(* Logix 5000 project; controller PRG_SPECK Emulate 5570 rev 30.12; software revision 30.00 *)

TASK MainTask (continuous, watchdog 5000 ms) : MainProgram

MODULES
   Local : Emulate 5570 (ICP 3, rev 30.12)
       : vendor 1 type 0 code 15 (ICP 0, rev 1.1, Output RPI 50 ms)
END_MODULES

TYPE UDT_BA :
STRUCT
   AL : BOOL;
END_STRUCT
END_TYPE

PROGRAM MainProgram   (* main routine MainRoutine *)
VAR
   PRG_Counter : DINT[2];
   PRG_i : DINT;
   PRG_j : DINT;
   PRG_Res_Len : DINT;
   PRG_Result : DINT[256];
   SCAN_CYCLE_TIME : DINT;
   Speck_AS_res : DINT[2];
   Speck_AS_tmp : DINT;
   Speck_AS_X : DINT[2] := ([0] := -536870912);
   Speck_AS_Y : DINT[2] := ([0] := 1610612736);
   Speck_Block_size : DINT;
   Speck_Carry_Bit : DINT;
   Speck_Ciphertext : DINT[2,2];
   Speck_dec_i : DINT;
   Speck_dec_j : DINT;
   Speck_enc_i : DINT;
   Speck_enc_j : DINT;
   Speck_i : DINT;
   Speck_j : DINT;
   Speck_key_size : DINT;
   Speck_Plaintext : DINT[2,2];
   Speck_Rd_Max : DINT;
   Speck_Rotate_Result : DINT[2];
   Speck_Round_Keys : DINT[34,2];
   Speck_Sign_Bits : DINT[2];
   Speck_tmp : DINT;
   Speck_tmp1 : DINT;
   Speck_tmp2 : DINT[2];
   Speck_Ver : DINT;
   Speck_x : DINT[2];
   Speck_y : DINT[2];
END_VAR

ROUTINE MainRoutine   (* ladder *)
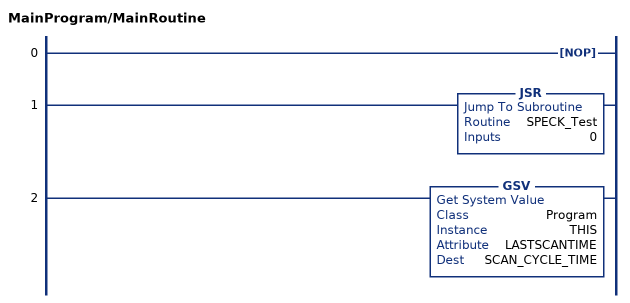
   0: NOP();
   1: JSR(SPECK_Test,0);
   2: GSV(Program,THIS,LASTSCANTIME,SCAN_CYCLE_TIME);
END_ROUTINE

ROUTINE PRG_PRF_Init   (* structured text *)
   //initialize version
   
   Speck_Ver:=2;     // 0: 32/64, 1: 64: 96, 2: 64:128, 3:128/128, 4:128/192, 5: 128/256
   
   PRG_j:=0;
   PRG_Res_Len :=  (PRG_Counter[0] AND 16#0000ffff)-1;
   
   JSR(SPECK_Init);
END_ROUTINE

ROUTINE PRG_PRF_SPECK   (* structured text *)
   // init PRG_Count[0] and PRG_Count[1] during application.. for PRF.. they could be any values
   //For PRG application, PRG_Count[0] defines the output length (i.e., the number of 64-bit, e.g., 128-bit output, PRG_Count[0]:=2)
   
   
   JSR(PRG_PRF_Init);
   
   PRG_j:=0;
   For PRG_i:=0 to PRG_Res_Len by 1 do
   	Speck_Plaintext[0,0]:=PRG_Counter[0]; //Upper bits of current plaintext
   	Speck_Plaintext[1,0]:=PRG_Counter[1];  //Lower bits of current plaintext
   	JSR(SPECK_Enc);
   	PRG_Result[PRG_j]:=Speck_Ciphertext[0,0];
   	PRG_Result[PRG_j+1]:=Speck_Ciphertext[1,0];
   
   	PRG_j:=PRG_j+2;
   
   End_For;
   
   JSR(SPECK_ClearKey);
   
END_ROUTINE

ROUTINE PRG_PRF_SPECK_Test   (* structured text *)
   
   //initialize version
   If S:FS Then
   
   	PRG_Counter[0]:=5;
   	PRG_Counter[1]:=1;
   
   
   End_if;
   
   
   JSR(PRG_PRF_SPECK);
END_ROUTINE

ROUTINE SPECK_Add   (* structured text *)
   	//big addition low 32-bit
   Speck_AS_res[0]:=0;
   Speck_AS_res[1]:=0;
   		Speck_Sign_Bits[0].[0]:= Speck_AS_X[0].30; //keep the sign bit for big addition
   		Speck_Sign_Bits[0].[1]:= Speck_AS_X[0].31;
   		Speck_AS_X[0].31:=0;
   		Speck_AS_X[0].30:=0;
   
   
   
   		Speck_Sign_Bits[1].[0]:= Speck_AS_Y[0].30; //keep the sign bit for big addition
   		Speck_Sign_Bits[1].[1]:= Speck_AS_Y[0].31;
   		Speck_AS_Y[0].31:=0;
   		Speck_AS_Y[0].30:=0;
   
   		Speck_AS_res[0] := Speck_AS_X[0]+Speck_AS_Y[0];
   
   		Speck_Carry_Bit.[0]:= Speck_AS_res[0].30;
   
   		Speck_AS_tmp:=Speck_Sign_Bits[1]+Speck_Sign_Bits[0]+Speck_Carry_Bit;
   
   		Speck_AS_res[0].[30]:= Speck_AS_tmp.[0];
   		Speck_AS_res[0].[31]:= Speck_AS_tmp.[1];
   
   		Speck_Carry_Bit.[0]:= Speck_AS_tmp.[2];
   
   
   		Speck_AS_tmp:=0;
   		Speck_Sign_Bits[0]:=0;
   		Speck_Sign_Bits[1]:=0;
   
   //add high 32-bit
   if Speck_Ver>2 then
   		Speck_Sign_Bits[0].[0]:= Speck_AS_X[1].30; //keep the sign bit for big addition
   		Speck_Sign_Bits[0].[1]:= Speck_AS_X[1].31;
   		Speck_AS_X[1].31:=0;
   		Speck_AS_X[1].30:=0;
   
   
   
   		Speck_Sign_Bits[1].[0]:= Speck_AS_Y[1].30; //keep the sign bit for big addition
   		Speck_Sign_Bits[1].[1]:= Speck_AS_Y[1].31;
   		Speck_AS_Y[1].31:=0;
   		Speck_AS_Y[1].30:=0;
   
   
   		Speck_AS_res[1]:=Speck_AS_X[1]+Speck_AS_Y[1]+Speck_Carry_Bit;
   
   		Speck_Carry_Bit.[0]:= Speck_AS_res[1].30;
   
   		Speck_AS_tmp:=Speck_Sign_Bits[1]+Speck_Sign_Bits[0]+Speck_Carry_Bit;
   
   		Speck_AS_res[1].[30]:= Speck_AS_tmp.[0];
   		Speck_AS_res[1].[31]:= Speck_AS_tmp.[1];
   
   end_if;
   
   
   		//clear
   		Speck_Carry_Bit:=0;
   		Speck_AS_tmp:=0;
   		Speck_Sign_Bits[0]:=0;
   		Speck_Sign_Bits[1]:=0;
   		Speck_AS_X[0]:=0;
   		Speck_AS_X[1]:=0;
   		Speck_AS_Y[0]:=0;
   		Speck_AS_Y[1]:=0;
   
   
END_ROUTINE

ROUTINE SPECK_ClearKey   (* structured text *)
   
   Speck_Round_Keys[0,0]:=0;
   Speck_Round_Keys[1,0]:=0;
   Speck_Round_Keys[2,0]:=0;
   Speck_Round_Keys[3,0]:=0;
   Speck_Round_Keys[4,0]:=0;
   Speck_Round_Keys[5,0]:=0;
   Speck_Round_Keys[6,0]:=0;
   Speck_Round_Keys[7,0]:=0;
   Speck_Round_Keys[8,0]:=0;
   Speck_Round_Keys[9,0]:=0;
   Speck_Round_Keys[10,0]:=0;
   Speck_Round_Keys[11,0]:=0;
   Speck_Round_Keys[12,0]:=0;
   Speck_Round_Keys[13,0]:=0;
   Speck_Round_Keys[14,0]:=0;
   Speck_Round_Keys[15,0]:=0;
   Speck_Round_Keys[16,0]:=0;
   Speck_Round_Keys[17,0]:=0;
   Speck_Round_Keys[18,0]:=0;
   Speck_Round_Keys[19,0]:=0;
   Speck_Round_Keys[20,0]:=0;
   Speck_Round_Keys[21,0]:=0;
   Speck_Round_Keys[22,0]:=0;
   Speck_Round_Keys[23,0]:=0;
   Speck_Round_Keys[24,0]:=0;
   Speck_Round_Keys[25,0]:=0;
   Speck_Round_Keys[26,0]:=0;
END_ROUTINE

ROUTINE SPECK_Dec   (* structured text *)
   
   JSR(SPECK_Init);
   
   
   
   
   Case Speck_Ver Of
   
   0,1,2:
   	Speck_Plaintext[0,0]:=Speck_Ciphertext[0,0];
   	Speck_Plaintext[1,0]:=Speck_Ciphertext[1,0];
   
   	For Speck_i:=Speck_Rd_Max to 0 by -1 do
   
   		Speck_AS_res[0]:= Speck_Plaintext[1,0] XOR Speck_Plaintext[0,0];
   
   		Speck_tmp2[0]:=Speck_AS_res[0];
   		JSR(SPECK_Rotate_Right_Dec);      //rotate based on Speck_AS_res[0]
   
   		Speck_Plaintext[0,0]:= Speck_Rotate_Result[0];
   
   		Speck_AS_X[0]:= Speck_Plaintext[1,0] XOR Speck_Round_Keys[Speck_i,0];
   
   
   
   		if Speck_Ver=0 Then
   			Speck_AS_X[0].16:=1;
   			Speck_AS_res[0]:= (Speck_AS_X[0]- Speck_Plaintext[0,0]) AND 16#0000ffff; //??AND 16#ffff;
   		Else
   			Speck_AS_Y[0]:=Speck_Plaintext[0,0];
   			JSR(SPECK_Sub);
   		End_if;
   		Speck_tmp2[0]:=Speck_AS_res[0];
   		JSR(SPECK_Rotate_Left_Dec);      //rotate based on Speck_AS_res[0]
   		Speck_Plaintext[1,0]:=Speck_Rotate_Result[0];
   
   	End_for;
   
   3,4,5:
   	Speck_Plaintext[0,0]:=Speck_Ciphertext[0,0];
   	Speck_Plaintext[0,1]:=Speck_Ciphertext[0,1];
   	Speck_Plaintext[1,0]:=Speck_Ciphertext[1,0];
   	Speck_Plaintext[1,1]:=Speck_Ciphertext[1,1];
   
   	For Speck_i:=Speck_Rd_Max to 0 by -1 do
   
   		Speck_AS_res[0]:= Speck_Plaintext[0,0] XOR Speck_Plaintext[1,0];
   		Speck_AS_res[1]:= Speck_Plaintext[0,1] XOR Speck_Plaintext[1,1];
   
   
   		Speck_tmp2[0]:=Speck_AS_res[0];
   		Speck_tmp2[1]:=Speck_AS_res[1];
   		JSR(SPECK_Rotate_Right_Dec);      //rotate based on Speck_AS_res[0] and Speck_AS_res[1]
   
   		Speck_Plaintext[0,0]:= Speck_Rotate_Result[0];
   		Speck_Plaintext[0,1]:= Speck_Rotate_Result[1];
   
   		Speck_AS_X[0]:= Speck_Plaintext[1,0] XOR Speck_Round_Keys[Speck_i,0];
   		Speck_AS_X[1]:= Speck_Plaintext[1,1] XOR Speck_Round_Keys[Speck_i,1];
   
   
   		Speck_AS_Y[0]:=Speck_Plaintext[0,0];
   		Speck_AS_Y[1]:=Speck_Plaintext[0,1];
   		JSR(SPECK_Sub);
   
   		Speck_tmp2[0]:=Speck_AS_res[0];
   		Speck_tmp2[1]:=Speck_AS_res[1];
   		JSR(SPECK_Rotate_Left_Dec);      //rotate based on Speck_AS_res[0] and Speck_AS_res[1]
   		Speck_Plaintext[1,0]:=Speck_Rotate_Result[0];
   		Speck_Plaintext[1,1]:=Speck_Rotate_Result[1];
   	End_for;
   
   End_Case;
   
   
   
   
   
   
   JSR(SPECK_ClearKey);
   
   
   
   
   
   
   
   
END_ROUTINE

ROUTINE SPECK_Enc   (* structured text *)
   
   Case Speck_Ver Of
   
   0,1,2:
   	Speck_Ciphertext[0,0]:=Speck_Plaintext[0,0];
   	Speck_Ciphertext[1,0]:=Speck_Plaintext[1,0];
   
   	For Speck_i:=0 to Speck_Rd_Max by 1 do
   		Speck_tmp2[0]:=Speck_Ciphertext[1,0];
   		JSR(SPECK_Rotate_Right_Enc);       //c1>>>>
   
   
   
   
   		if Speck_Ver=0 Then
   			Speck_Ciphertext[1,0]:= (Speck_Rotate_Result[0] + Speck_Ciphertext[0,0]) XOR Speck_Round_Keys[Speck_i,0];
   			Speck_Ciphertext[1,0]:= Speck_Ciphertext[1,0] AND 16#0000ffff;
   		Else
   			Speck_AS_X[0]:=Speck_Rotate_Result[0];
   			Speck_AS_Y[0]:=Speck_Ciphertext[0,0];
   			JSR(SPECK_Add);
   			Speck_Ciphertext[1,0]:= Speck_AS_res[0] XOR Speck_Round_Keys[Speck_i,0];
   		End_if;
   
   
   		Speck_tmp2[0]:=Speck_Ciphertext[0,0];
   		JSR(SPECK_Rotate_Left_Enc);   //p0<<<
   		Speck_Ciphertext[0,0]:=Speck_Rotate_Result[0] XOR Speck_Ciphertext[1,0];
   	End_for;
   
   3,4,5:
   	Speck_Ciphertext[0,0]:=Speck_Plaintext[0,0];
   	Speck_Ciphertext[0,1]:=Speck_Plaintext[0,1];
   	Speck_Ciphertext[1,0]:=Speck_Plaintext[1,0];
   	Speck_Ciphertext[1,1]:=Speck_Plaintext[1,1];
   
   	For Speck_i:=0 to Speck_Rd_Max by 1 do
   		Speck_tmp2[0]:=Speck_Ciphertext[1,0];
   		Speck_tmp2[1]:=Speck_Ciphertext[1,1];
   		JSR(SPECK_Rotate_Right_Enc);       //c1>>>>
   
   
   
   
   		Speck_AS_X[0]:=Speck_Rotate_Result[0];
   		Speck_AS_X[1]:=Speck_Rotate_Result[1];
   		Speck_AS_Y[0]:=Speck_Ciphertext[0,0];
   		Speck_AS_Y[1]:=Speck_Ciphertext[0,1];
   		JSR(SPECK_Add);
   		Speck_Ciphertext[1,0]:= Speck_AS_res[0] XOR Speck_Round_Keys[Speck_i,0];
   	 	Speck_Ciphertext[1,1]:= Speck_AS_res[1] XOR Speck_Round_Keys[Speck_i,1];
   
   
   		Speck_tmp2[0]:=Speck_Ciphertext[0,0];
   		Speck_tmp2[1]:=Speck_Ciphertext[0,1];
   		JSR(SPECK_Rotate_Left_Enc);   //c0<<<
   		Speck_Ciphertext[0,0]:=Speck_Rotate_Result[0] XOR Speck_Ciphertext[1,0];
   		Speck_Ciphertext[0,1]:=Speck_Rotate_Result[1] XOR Speck_Ciphertext[1,1];
   	End_for;
   
   End_Case;
   
   
   
   
   
   JSR(SPECK_ClearKey);
   
   
   
   
   
   
END_ROUTINE

ROUTINE SPECK_Init   (* structured text *)
   CASE Speck_Ver Of
   	0:
   		//Speck_Rd_Max:=21;
   		Speck_Rd_Max:=21;
   		Speck_Round_Keys[0,0]:=15631;
   		//Speck_Round_Keys[0,0]:=0;
   		Speck_Round_Keys[1,0]:=9700;
   		Speck_Round_Keys[2,0]:=61996;
   		Speck_Round_Keys[3,0]:=19213;
   		Speck_Round_Keys[4,0]:=12568;
   		Speck_Round_Keys[5,0]:=53935;
   		Speck_Round_Keys[6,0]:=268;
   		Speck_Round_Keys[7,0]:=50664;
   		Speck_Round_Keys[8,0]:=60120;
   		Speck_Round_Keys[9,0]:=40333;
   		Speck_Round_Keys[10,0]:=24732;
   		Speck_Round_Keys[11,0]:=23055;
   		Speck_Round_Keys[12,0]:=43006;
   		Speck_Round_Keys[13,0]:=3801;
   		Speck_Round_Keys[14,0]:=54139;
   		Speck_Round_Keys[15,0]:=30112;
   		Speck_Round_Keys[16,0]:=55913;
   		Speck_Round_Keys[17,0]:=28143;
   		Speck_Round_Keys[18,0]:=63915;
   		Speck_Round_Keys[19,0]:=1151;
   		Speck_Round_Keys[20,0]:=48927;
   		Speck_Round_Keys[21,0]:=23424;
   	1:
   		Speck_Rd_Max:=25;
   		Speck_Round_Keys[0,0]:=1010479052;
   		Speck_Round_Keys[1,0]:=1960303416;
   		Speck_Round_Keys[2,0]:=1299975900;
   		Speck_Round_Keys[3,0]:=-1898951853;
   		Speck_Round_Keys[4,0]:=-1343771839;
   		Speck_Round_Keys[5,0]:=1072967228;
   		Speck_Round_Keys[6,0]:=1891935448;
   		Speck_Round_Keys[7,0]:=-862191615;
   		Speck_Round_Keys[8,0]:=-24294679;
   		Speck_Round_Keys[9,0]:=1209777;
   		Speck_Round_Keys[10,0]:=-379647130;
   		Speck_Round_Keys[11,0]:=-429531458;
   		Speck_Round_Keys[12,0]:=1219013850;
   		Speck_Round_Keys[13,0]:=1258773305;
   		Speck_Round_Keys[14,0]:=1958978832;
   		Speck_Round_Keys[15,0]:=-1299080388;
   		Speck_Round_Keys[16,0]:=1521232504;
   		Speck_Round_Keys[17,0]:=-1755465132;
   		Speck_Round_Keys[18,0]:=-1183209214;
   		Speck_Round_Keys[19,0]:=-497510761;
   		Speck_Round_Keys[20,0]:=-65018188;
   		Speck_Round_Keys[21,0]:=627271131;
   		Speck_Round_Keys[22,0]:=289351083;
   		Speck_Round_Keys[23,0]:=163990315;
   		Speck_Round_Keys[24,0]:=-1174022665;
   		Speck_Round_Keys[25,0]:=-1342639090;
   	2:
   		Speck_Rd_Max:=26;
   		Speck_Round_Keys[0,0]:=-1148848103;
   		Speck_Round_Keys[1,0]:=1208089977;
   		Speck_Round_Keys[2,0]:=-1783362989;
   		Speck_Round_Keys[3,0]:=-914269261;
   		Speck_Round_Keys[4,0]:=-1304315992;
   		Speck_Round_Keys[5,0]:=-2127551690;
   		Speck_Round_Keys[6,0]:=-823047894;
   		Speck_Round_Keys[7,0]:=-1124290961;
   		Speck_Round_Keys[8,0]:=-2081609188;
   		Speck_Round_Keys[9,0]:=-1368174669;
   		Speck_Round_Keys[10,0]:=1254090106;
   		Speck_Round_Keys[11,0]:=-1215402569;
   		Speck_Round_Keys[12,0]:=-1522370332;
   		Speck_Round_Keys[13,0]:=-9254945;
   		Speck_Round_Keys[14,0]:=-770318043;
   		Speck_Round_Keys[15,0]:=-1248627894;
   		Speck_Round_Keys[16,0]:=1667665164;
   		Speck_Round_Keys[17,0]:=1127551330;
   		Speck_Round_Keys[18,0]:=1631463370;
   		Speck_Round_Keys[19,0]:=339858424;
   		Speck_Round_Keys[20,0]:=1104564693;
   		Speck_Round_Keys[21,0]:=-1092140090;
   		Speck_Round_Keys[22,0]:=-34819784;
   		Speck_Round_Keys[23,0]:=-1239678853;
   		Speck_Round_Keys[24,0]:=1539057967;
   		Speck_Round_Keys[25,0]:=1646443297;
   		Speck_Round_Keys[26,0]:=99633891;
   	3:
   		Speck_Rd_Max:=31;
   		Speck_Round_Keys[0,0]:=-2080825868;
   		Speck_Round_Keys[0,1]:=-649265456;
   		Speck_Round_Keys[1,0]:=2050826354;
   		Speck_Round_Keys[1,1]:=789043958;
   		Speck_Round_Keys[2,0]:=1076159464;
   		Speck_Round_Keys[2,1]:=1207346796;
   		Speck_Round_Keys[3,0]:=-1868617995;
   		Speck_Round_Keys[3,1]:=27785654;
   		Speck_Round_Keys[4,0]:=653389667;
   		Speck_Round_Keys[4,1]:=857678648;
   		Speck_Round_Keys[5,0]:=1480341691;
   		Speck_Round_Keys[5,1]:=-1263296287;
   		Speck_Round_Keys[6,0]:=-1964153065;
   		Speck_Round_Keys[6,1]:=-1671577777;
   		Speck_Round_Keys[7,0]:=862328600;
   		Speck_Round_Keys[7,1]:=2036511554;
   		Speck_Round_Keys[8,0]:=81192154;
   		Speck_Round_Keys[8,1]:=-687588873;
   		Speck_Round_Keys[9,0]:=-1917483227;
   		Speck_Round_Keys[9,1]:=63249243;
   		Speck_Round_Keys[10,0]:=-1952596082;
   		Speck_Round_Keys[10,1]:=2143544786;
   		Speck_Round_Keys[11,0]:=-1544920938;
   		Speck_Round_Keys[11,1]:=1465879784;
   		Speck_Round_Keys[12,0]:=2139891583;
   		Speck_Round_Keys[12,1]:=1710163122;
   		Speck_Round_Keys[13,0]:=-1608051307;
   		Speck_Round_Keys[13,1]:=-1374801591;
   		Speck_Round_Keys[14,0]:=943121719;
   		Speck_Round_Keys[14,1]:=354429694;
   		Speck_Round_Keys[15,0]:=582741445;
   		Speck_Round_Keys[15,1]:=-2054972675;
   		Speck_Round_Keys[16,0]:=1721968636;
   		Speck_Round_Keys[16,1]:=-1512022332;
   		Speck_Round_Keys[17,0]:=-1725680323;
   		Speck_Round_Keys[17,1]:=1657126074;
   		Speck_Round_Keys[18,0]:=247339174;
   		Speck_Round_Keys[18,1]:=1221108278;
   		Speck_Round_Keys[19,0]:=-807872440;
   		Speck_Round_Keys[19,1]:=-1429436100;
   		Speck_Round_Keys[20,0]:=1418166873;
   		Speck_Round_Keys[20,1]:=-215130835;
   		Speck_Round_Keys[21,0]:=-621280229;
   		Speck_Round_Keys[21,1]:=412315805;
   		Speck_Round_Keys[22,0]:=1459956154;
   		Speck_Round_Keys[22,1]:=-1758754260;
   		Speck_Round_Keys[23,0]:=435300123;
   		Speck_Round_Keys[23,1]:=-1545364290;
   		Speck_Round_Keys[24,0]:=1027574508;
   		Speck_Round_Keys[24,1]:=-481319156;
   		Speck_Round_Keys[25,0]:=1691703329;
   		Speck_Round_Keys[25,1]:=651500257;
   		Speck_Round_Keys[26,0]:=1740505566;
   		Speck_Round_Keys[26,1]:=1823342560;
   		Speck_Round_Keys[27,0]:=1022031660;
   		Speck_Round_Keys[27,1]:=749650446;
   		Speck_Round_Keys[28,0]:=-397311955;
   		Speck_Round_Keys[28,1]:=83994786;
   		Speck_Round_Keys[29,0]:=800982389;
   		Speck_Round_Keys[29,1]:=-646252930;
   		Speck_Round_Keys[30,0]:=1439684980;
   		Speck_Round_Keys[30,1]:=386814096;
   		Speck_Round_Keys[31,0]:=-873348581;
   		Speck_Round_Keys[31,1]:=-1190976360;
   	4:
   		Speck_Rd_Max:=32;
   		Speck_Round_Keys[0,0]:=-2109044216;
   		Speck_Round_Keys[0,1]:=-434844049;
   		Speck_Round_Keys[1,0]:=-1420570460;
   		Speck_Round_Keys[1,1]:=2000435062;
   		Speck_Round_Keys[2,0]:=663289456;
   		Speck_Round_Keys[2,1]:=-1180846514;
   		Speck_Round_Keys[3,0]:=1579651993;
   		Speck_Round_Keys[3,1]:=66732943;
   		Speck_Round_Keys[4,0]:=-949825977;
   		Speck_Round_Keys[4,1]:=-1943390162;
   		Speck_Round_Keys[5,0]:=586375629;
   		Speck_Round_Keys[5,1]:=992192424;
   		Speck_Round_Keys[6,0]:=805843267;
   		Speck_Round_Keys[6,1]:=1590578209;
   		Speck_Round_Keys[7,0]:=-1864178662;
   		Speck_Round_Keys[7,1]:=-488374217;
   		Speck_Round_Keys[8,0]:=1152511586;
   		Speck_Round_Keys[8,1]:=-194034418;
   		Speck_Round_Keys[9,0]:=-916674430;
   		Speck_Round_Keys[9,1]:=510305946;
   		Speck_Round_Keys[10,0]:=61438023;
   		Speck_Round_Keys[10,1]:=-443574147;
   		Speck_Round_Keys[11,0]:=1283870034;
   		Speck_Round_Keys[11,1]:=1171556711;
   		Speck_Round_Keys[12,0]:=-1044183024;
   		Speck_Round_Keys[12,1]:=1485368022;
   		Speck_Round_Keys[13,0]:=60705369;
   		Speck_Round_Keys[13,1]:=1673274192;
   		Speck_Round_Keys[14,0]:=181714170;
   		Speck_Round_Keys[14,1]:=-810971494;
   		Speck_Round_Keys[15,0]:=-1452546250;
   		Speck_Round_Keys[15,1]:=-2049570575;
   		Speck_Round_Keys[16,0]:=563980564;
   		Speck_Round_Keys[16,1]:=1508672253;
   		Speck_Round_Keys[17,0]:=-1726885166;
   		Speck_Round_Keys[17,1]:=1988838192;
   		Speck_Round_Keys[18,0]:=-11526877;
   		Speck_Round_Keys[18,1]:=-1858736650;
   		Speck_Round_Keys[19,0]:=-963990845;
   		Speck_Round_Keys[19,1]:=-817492171;
   		Speck_Round_Keys[20,0]:=1478577398;
   		Speck_Round_Keys[20,1]:=-1380080500;
   		Speck_Round_Keys[21,0]:=-1676330340;
   		Speck_Round_Keys[21,1]:=1534823287;
   		Speck_Round_Keys[22,0]:=-2026497924;
   		Speck_Round_Keys[22,1]:=-1854221332;
   		Speck_Round_Keys[23,0]:=1666823377;
   		Speck_Round_Keys[23,1]:=1853488750;
   		Speck_Round_Keys[24,0]:=-158124369;
   		Speck_Round_Keys[24,1]:=-1736367530;
   		Speck_Round_Keys[25,0]:=1832056096;
   		Speck_Round_Keys[25,1]:=-709491608;
   		Speck_Round_Keys[26,0]:=-1320038234;
   		Speck_Round_Keys[26,1]:=-946880541;
   		Speck_Round_Keys[27,0]:=-2048989650;
   		Speck_Round_Keys[27,1]:=1069091871;
   		Speck_Round_Keys[28,0]:=-1081468659;
   		Speck_Round_Keys[28,1]:=493915857;
   		Speck_Round_Keys[29,0]:=1244604632;
   		Speck_Round_Keys[29,1]:=209165789;
   		Speck_Round_Keys[30,0]:=-516878538;
   		Speck_Round_Keys[30,1]:=967074394;
   		Speck_Round_Keys[31,0]:=528572285;
   		Speck_Round_Keys[31,1]:=-27129480;
   		Speck_Round_Keys[32,0]:=-1066840277;
   		Speck_Round_Keys[32,1]:=-1998704319;
   	5:
   		Speck_Rd_Max:=33;
   		//Speck_Rd_Max:=0;
   		Speck_Round_Keys[0,0]:=-1203303343;
   		Speck_Round_Keys[0,1]:=1330976216;
   		Speck_Round_Keys[1,0]:=1407326483;
   		Speck_Round_Keys[1,1]:=-1724620941;
   		Speck_Round_Keys[2,0]:=-1336357073;
   		Speck_Round_Keys[2,1]:=2075201973;
   		Speck_Round_Keys[3,0]:=-1964127817;
   		Speck_Round_Keys[3,1]:=-1676860110;
   		Speck_Round_Keys[4,0]:=-2129443066;
   		Speck_Round_Keys[4,1]:=1324272631;
   		Speck_Round_Keys[5,0]:=-1616999486;
   		Speck_Round_Keys[5,1]:=1032033716;
   		Speck_Round_Keys[6,0]:=238450941;
   		Speck_Round_Keys[6,1]:=454117302;
   		Speck_Round_Keys[7,0]:=-2133053345;
   		Speck_Round_Keys[7,1]:=2016900436;
   		Speck_Round_Keys[8,0]:=1979592355;
   		Speck_Round_Keys[8,1]:=-1585551365;
   		Speck_Round_Keys[9,0]:=1247927760;
   		Speck_Round_Keys[9,1]:=559820155;
   		Speck_Round_Keys[10,0]:=2074240269;
   		Speck_Round_Keys[10,1]:=1096187537;
   		Speck_Round_Keys[11,0]:=-1544710491;
   		Speck_Round_Keys[11,1]:=-971052382;
   		Speck_Round_Keys[12,0]:=1614561484;
   		Speck_Round_Keys[12,1]:=-1118146933;
   		Speck_Round_Keys[13,0]:=625176544;
   		Speck_Round_Keys[13,1]:=-1517436671;
   		Speck_Round_Keys[14,0]:=-1440617253;
   		Speck_Round_Keys[14,1]:=-1662713437;
   		Speck_Round_Keys[15,0]:=503283530;
   		Speck_Round_Keys[15,1]:=1995145044;
   		Speck_Round_Keys[16,0]:=284729323;
   		Speck_Round_Keys[16,1]:=-825926335;
   		Speck_Round_Keys[17,0]:=1430104656;
   		Speck_Round_Keys[17,1]:=-1991245376;
   		Speck_Round_Keys[18,0]:=294868347;
   		Speck_Round_Keys[18,1]:=-458348607;
   		Speck_Round_Keys[19,0]:=1158525600;
   		Speck_Round_Keys[19,1]:=601377666;
   		Speck_Round_Keys[20,0]:=1936684124;
   		Speck_Round_Keys[20,1]:=1623592388;
   		Speck_Round_Keys[21,0]:=1182373476;
   		Speck_Round_Keys[21,1]:=795858385;
   		Speck_Round_Keys[22,0]:=-1645874420;
   		Speck_Round_Keys[22,1]:=755343120;
   		Speck_Round_Keys[23,0]:=1526816951;
   		Speck_Round_Keys[23,1]:=247936705;
   		Speck_Round_Keys[24,0]:=2013201414;
   		Speck_Round_Keys[24,1]:=-80764261;
   		Speck_Round_Keys[25,0]:=326734656;
   		Speck_Round_Keys[25,1]:=-857819692;
   		Speck_Round_Keys[26,0]:=22458222;
   		Speck_Round_Keys[26,1]:=1789592334;
   		Speck_Round_Keys[27,0]:=-53318718;
   		Speck_Round_Keys[27,1]:=2100444963;
   		Speck_Round_Keys[28,0]:=-31841512;
   		Speck_Round_Keys[28,1]:=-838605044;
   		Speck_Round_Keys[29,0]:=-1477810343;
   		Speck_Round_Keys[29,1]:=-1127145226;
   		Speck_Round_Keys[30,0]:=-1047355237;
   		Speck_Round_Keys[30,1]:=-232830838;
   		Speck_Round_Keys[31,0]:=842943118;
   		Speck_Round_Keys[31,1]:=1252680607;
   		Speck_Round_Keys[32,0]:=-1978168146;
   		Speck_Round_Keys[32,1]:=2089790505;
   		Speck_Round_Keys[33,0]:=1886440712;
   		Speck_Round_Keys[33,1]:=1660119865;
   End_CASE;
   
END_ROUTINE

ROUTINE SPECK_Rotate_Left_Dec   (* structured text *)
   Speck_Rotate_Result[0]:=0;
   Speck_Rotate_Result[1]:=0;
   
   CASE Speck_Ver Of
   	0:
   		Speck_Rotate_Result[0].[6]:=Speck_tmp2[0].[15];
   		Speck_Rotate_Result[0].[5]:=Speck_tmp2[0].[14];
   		Speck_Rotate_Result[0].[4]:=Speck_tmp2[0].[13];
   		Speck_Rotate_Result[0].[3]:=Speck_tmp2[0].[12];
   		Speck_Rotate_Result[0].[2]:=Speck_tmp2[0].[11];
   		Speck_Rotate_Result[0].[1]:=Speck_tmp2[0].[10];
   		Speck_Rotate_Result[0].[0]:=Speck_tmp2[0].[9];
   		Speck_Rotate_Result[0].[15]:=Speck_tmp2[0].[8];
   		Speck_Rotate_Result[0].[14]:=Speck_tmp2[0].[7];
   		Speck_Rotate_Result[0].[13]:=Speck_tmp2[0].[6];
   		Speck_Rotate_Result[0].[12]:=Speck_tmp2[0].[5];
   		Speck_Rotate_Result[0].[11]:=Speck_tmp2[0].[4];
   		Speck_Rotate_Result[0].[10]:=Speck_tmp2[0].[3];
   		Speck_Rotate_Result[0].[9]:=Speck_tmp2[0].[2];
   		Speck_Rotate_Result[0].[8]:=Speck_tmp2[0].[1];
   		Speck_Rotate_Result[0].[7]:=Speck_tmp2[0].[0];
   	1,2:
   		Speck_Rotate_Result[0].[7]:=Speck_tmp2[0].[31];
   		Speck_Rotate_Result[0].[6]:=Speck_tmp2[0].[30];
   		Speck_Rotate_Result[0].[5]:=Speck_tmp2[0].[29];
   		Speck_Rotate_Result[0].[4]:=Speck_tmp2[0].[28];
   		Speck_Rotate_Result[0].[3]:=Speck_tmp2[0].[27];
   		Speck_Rotate_Result[0].[2]:=Speck_tmp2[0].[26];
   		Speck_Rotate_Result[0].[1]:=Speck_tmp2[0].[25];
   		Speck_Rotate_Result[0].[0]:=Speck_tmp2[0].[24];
   		Speck_Rotate_Result[0].[31]:=Speck_tmp2[0].[23];
   		Speck_Rotate_Result[0].[30]:=Speck_tmp2[0].[22];
   		Speck_Rotate_Result[0].[29]:=Speck_tmp2[0].[21];
   		Speck_Rotate_Result[0].[28]:=Speck_tmp2[0].[20];
   		Speck_Rotate_Result[0].[27]:=Speck_tmp2[0].[19];
   		Speck_Rotate_Result[0].[26]:=Speck_tmp2[0].[18];
   		Speck_Rotate_Result[0].[25]:=Speck_tmp2[0].[17];
   		Speck_Rotate_Result[0].[24]:=Speck_tmp2[0].[16];
   		Speck_Rotate_Result[0].[23]:=Speck_tmp2[0].[15];
   		Speck_Rotate_Result[0].[22]:=Speck_tmp2[0].[14];
   		Speck_Rotate_Result[0].[21]:=Speck_tmp2[0].[13];
   		Speck_Rotate_Result[0].[20]:=Speck_tmp2[0].[12];
   		Speck_Rotate_Result[0].[19]:=Speck_tmp2[0].[11];
   		Speck_Rotate_Result[0].[18]:=Speck_tmp2[0].[10];
   		Speck_Rotate_Result[0].[17]:=Speck_tmp2[0].[9];
   		Speck_Rotate_Result[0].[16]:=Speck_tmp2[0].[8];
   		Speck_Rotate_Result[0].[15]:=Speck_tmp2[0].[7];
   		Speck_Rotate_Result[0].[14]:=Speck_tmp2[0].[6];
   		Speck_Rotate_Result[0].[13]:=Speck_tmp2[0].[5];
   		Speck_Rotate_Result[0].[12]:=Speck_tmp2[0].[4];
   		Speck_Rotate_Result[0].[11]:=Speck_tmp2[0].[3];
   		Speck_Rotate_Result[0].[10]:=Speck_tmp2[0].[2];
   		Speck_Rotate_Result[0].[9]:=Speck_tmp2[0].[1];
   		Speck_Rotate_Result[0].[8]:=Speck_tmp2[0].[0];
   	3,4,5:
   		Speck_Rotate_Result[0].[7]:=Speck_tmp2[1].[31];
   		Speck_Rotate_Result[0].[6]:=Speck_tmp2[1].[30];
   		Speck_Rotate_Result[0].[5]:=Speck_tmp2[1].[29];
   		Speck_Rotate_Result[0].[4]:=Speck_tmp2[1].[28];
   		Speck_Rotate_Result[0].[3]:=Speck_tmp2[1].[27];
   		Speck_Rotate_Result[0].[2]:=Speck_tmp2[1].[26];
   		Speck_Rotate_Result[0].[1]:=Speck_tmp2[1].[25];
   		Speck_Rotate_Result[0].[0]:=Speck_tmp2[1].[24];
   		Speck_Rotate_Result[1].[31]:=Speck_tmp2[1].[23];
   		Speck_Rotate_Result[1].[30]:=Speck_tmp2[1].[22];
   		Speck_Rotate_Result[1].[29]:=Speck_tmp2[1].[21];
   		Speck_Rotate_Result[1].[28]:=Speck_tmp2[1].[20];
   		Speck_Rotate_Result[1].[27]:=Speck_tmp2[1].[19];
   		Speck_Rotate_Result[1].[26]:=Speck_tmp2[1].[18];
   		Speck_Rotate_Result[1].[25]:=Speck_tmp2[1].[17];
   		Speck_Rotate_Result[1].[24]:=Speck_tmp2[1].[16];
   		Speck_Rotate_Result[1].[23]:=Speck_tmp2[1].[15];
   		Speck_Rotate_Result[1].[22]:=Speck_tmp2[1].[14];
   		Speck_Rotate_Result[1].[21]:=Speck_tmp2[1].[13];
   		Speck_Rotate_Result[1].[20]:=Speck_tmp2[1].[12];
   		Speck_Rotate_Result[1].[19]:=Speck_tmp2[1].[11];
   		Speck_Rotate_Result[1].[18]:=Speck_tmp2[1].[10];
   		Speck_Rotate_Result[1].[17]:=Speck_tmp2[1].[9];
   		Speck_Rotate_Result[1].[16]:=Speck_tmp2[1].[8];
   		Speck_Rotate_Result[1].[15]:=Speck_tmp2[1].[7];
   		Speck_Rotate_Result[1].[14]:=Speck_tmp2[1].[6];
   		Speck_Rotate_Result[1].[13]:=Speck_tmp2[1].[5];
   		Speck_Rotate_Result[1].[12]:=Speck_tmp2[1].[4];
   		Speck_Rotate_Result[1].[11]:=Speck_tmp2[1].[3];
   		Speck_Rotate_Result[1].[10]:=Speck_tmp2[1].[2];
   		Speck_Rotate_Result[1].[9]:=Speck_tmp2[1].[1];
   		Speck_Rotate_Result[1].[8]:=Speck_tmp2[1].[0];
   		Speck_Rotate_Result[1].[7]:=Speck_tmp2[0].[31];
   		Speck_Rotate_Result[1].[6]:=Speck_tmp2[0].[30];
   		Speck_Rotate_Result[1].[5]:=Speck_tmp2[0].[29];
   		Speck_Rotate_Result[1].[4]:=Speck_tmp2[0].[28];
   		Speck_Rotate_Result[1].[3]:=Speck_tmp2[0].[27];
   		Speck_Rotate_Result[1].[2]:=Speck_tmp2[0].[26];
   		Speck_Rotate_Result[1].[1]:=Speck_tmp2[0].[25];
   		Speck_Rotate_Result[1].[0]:=Speck_tmp2[0].[24];
   		Speck_Rotate_Result[0].[31]:=Speck_tmp2[0].[23];
   		Speck_Rotate_Result[0].[30]:=Speck_tmp2[0].[22];
   		Speck_Rotate_Result[0].[29]:=Speck_tmp2[0].[21];
   		Speck_Rotate_Result[0].[28]:=Speck_tmp2[0].[20];
   		Speck_Rotate_Result[0].[27]:=Speck_tmp2[0].[19];
   		Speck_Rotate_Result[0].[26]:=Speck_tmp2[0].[18];
   		Speck_Rotate_Result[0].[25]:=Speck_tmp2[0].[17];
   		Speck_Rotate_Result[0].[24]:=Speck_tmp2[0].[16];
   		Speck_Rotate_Result[0].[23]:=Speck_tmp2[0].[15];
   		Speck_Rotate_Result[0].[22]:=Speck_tmp2[0].[14];
   		Speck_Rotate_Result[0].[21]:=Speck_tmp2[0].[13];
   		Speck_Rotate_Result[0].[20]:=Speck_tmp2[0].[12];
   		Speck_Rotate_Result[0].[19]:=Speck_tmp2[0].[11];
   		Speck_Rotate_Result[0].[18]:=Speck_tmp2[0].[10];
   		Speck_Rotate_Result[0].[17]:=Speck_tmp2[0].[9];
   		Speck_Rotate_Result[0].[16]:=Speck_tmp2[0].[8];
   		Speck_Rotate_Result[0].[15]:=Speck_tmp2[0].[7];
   		Speck_Rotate_Result[0].[14]:=Speck_tmp2[0].[6];
   		Speck_Rotate_Result[0].[13]:=Speck_tmp2[0].[5];
   		Speck_Rotate_Result[0].[12]:=Speck_tmp2[0].[4];
   		Speck_Rotate_Result[0].[11]:=Speck_tmp2[0].[3];
   		Speck_Rotate_Result[0].[10]:=Speck_tmp2[0].[2];
   		Speck_Rotate_Result[0].[9]:=Speck_tmp2[0].[1];
   		Speck_Rotate_Result[0].[8]:=Speck_tmp2[0].[0];
   End_CASE;
   
END_ROUTINE

ROUTINE SPECK_Rotate_Left_Enc   (* structured text *)
   Speck_Rotate_Result[0]:=0;
   Speck_Rotate_Result[1]:=0;
   CASE Speck_Ver Of
   	0:
   		Speck_Rotate_Result[0].[1]:=Speck_tmp2[0].[15];
   		Speck_Rotate_Result[0].[0]:=Speck_tmp2[0].[14];
   		Speck_Rotate_Result[0].[15]:=Speck_tmp2[0].[13];
   		Speck_Rotate_Result[0].[14]:=Speck_tmp2[0].[12];
   		Speck_Rotate_Result[0].[13]:=Speck_tmp2[0].[11];
   		Speck_Rotate_Result[0].[12]:=Speck_tmp2[0].[10];
   		Speck_Rotate_Result[0].[11]:=Speck_tmp2[0].[9];
   		Speck_Rotate_Result[0].[10]:=Speck_tmp2[0].[8];
   		Speck_Rotate_Result[0].[9]:=Speck_tmp2[0].[7];
   		Speck_Rotate_Result[0].[8]:=Speck_tmp2[0].[6];
   		Speck_Rotate_Result[0].[7]:=Speck_tmp2[0].[5];
   		Speck_Rotate_Result[0].[6]:=Speck_tmp2[0].[4];
   		Speck_Rotate_Result[0].[5]:=Speck_tmp2[0].[3];
   		Speck_Rotate_Result[0].[4]:=Speck_tmp2[0].[2];
   		Speck_Rotate_Result[0].[3]:=Speck_tmp2[0].[1];
   		Speck_Rotate_Result[0].[2]:=Speck_tmp2[0].[0];
   	1,2:
   		Speck_Rotate_Result[0].[2]:=Speck_tmp2[0].[31];
   		Speck_Rotate_Result[0].[1]:=Speck_tmp2[0].[30];
   		Speck_Rotate_Result[0].[0]:=Speck_tmp2[0].[29];
   		Speck_Rotate_Result[0].[31]:=Speck_tmp2[0].[28];
   		Speck_Rotate_Result[0].[30]:=Speck_tmp2[0].[27];
   		Speck_Rotate_Result[0].[29]:=Speck_tmp2[0].[26];
   		Speck_Rotate_Result[0].[28]:=Speck_tmp2[0].[25];
   		Speck_Rotate_Result[0].[27]:=Speck_tmp2[0].[24];
   		Speck_Rotate_Result[0].[26]:=Speck_tmp2[0].[23];
   		Speck_Rotate_Result[0].[25]:=Speck_tmp2[0].[22];
   		Speck_Rotate_Result[0].[24]:=Speck_tmp2[0].[21];
   		Speck_Rotate_Result[0].[23]:=Speck_tmp2[0].[20];
   		Speck_Rotate_Result[0].[22]:=Speck_tmp2[0].[19];
   		Speck_Rotate_Result[0].[21]:=Speck_tmp2[0].[18];
   		Speck_Rotate_Result[0].[20]:=Speck_tmp2[0].[17];
   		Speck_Rotate_Result[0].[19]:=Speck_tmp2[0].[16];
   		Speck_Rotate_Result[0].[18]:=Speck_tmp2[0].[15];
   		Speck_Rotate_Result[0].[17]:=Speck_tmp2[0].[14];
   		Speck_Rotate_Result[0].[16]:=Speck_tmp2[0].[13];
   		Speck_Rotate_Result[0].[15]:=Speck_tmp2[0].[12];
   		Speck_Rotate_Result[0].[14]:=Speck_tmp2[0].[11];
   		Speck_Rotate_Result[0].[13]:=Speck_tmp2[0].[10];
   		Speck_Rotate_Result[0].[12]:=Speck_tmp2[0].[9];
   		Speck_Rotate_Result[0].[11]:=Speck_tmp2[0].[8];
   		Speck_Rotate_Result[0].[10]:=Speck_tmp2[0].[7];
   		Speck_Rotate_Result[0].[9]:=Speck_tmp2[0].[6];
   		Speck_Rotate_Result[0].[8]:=Speck_tmp2[0].[5];
   		Speck_Rotate_Result[0].[7]:=Speck_tmp2[0].[4];
   		Speck_Rotate_Result[0].[6]:=Speck_tmp2[0].[3];
   		Speck_Rotate_Result[0].[5]:=Speck_tmp2[0].[2];
   		Speck_Rotate_Result[0].[4]:=Speck_tmp2[0].[1];
   		Speck_Rotate_Result[0].[3]:=Speck_tmp2[0].[0];
   	3,4,5:
   		Speck_Rotate_Result[0].[2]:=Speck_tmp2[1].[31];
   		Speck_Rotate_Result[0].[1]:=Speck_tmp2[1].[30];
   		Speck_Rotate_Result[0].[0]:=Speck_tmp2[1].[29];
   		Speck_Rotate_Result[1].[31]:=Speck_tmp2[1].[28];
   		Speck_Rotate_Result[1].[30]:=Speck_tmp2[1].[27];
   		Speck_Rotate_Result[1].[29]:=Speck_tmp2[1].[26];
   		Speck_Rotate_Result[1].[28]:=Speck_tmp2[1].[25];
   		Speck_Rotate_Result[1].[27]:=Speck_tmp2[1].[24];
   		Speck_Rotate_Result[1].[26]:=Speck_tmp2[1].[23];
   		Speck_Rotate_Result[1].[25]:=Speck_tmp2[1].[22];
   		Speck_Rotate_Result[1].[24]:=Speck_tmp2[1].[21];
   		Speck_Rotate_Result[1].[23]:=Speck_tmp2[1].[20];
   		Speck_Rotate_Result[1].[22]:=Speck_tmp2[1].[19];
   		Speck_Rotate_Result[1].[21]:=Speck_tmp2[1].[18];
   		Speck_Rotate_Result[1].[20]:=Speck_tmp2[1].[17];
   		Speck_Rotate_Result[1].[19]:=Speck_tmp2[1].[16];
   		Speck_Rotate_Result[1].[18]:=Speck_tmp2[1].[15];
   		Speck_Rotate_Result[1].[17]:=Speck_tmp2[1].[14];
   		Speck_Rotate_Result[1].[16]:=Speck_tmp2[1].[13];
   		Speck_Rotate_Result[1].[15]:=Speck_tmp2[1].[12];
   		Speck_Rotate_Result[1].[14]:=Speck_tmp2[1].[11];
   		Speck_Rotate_Result[1].[13]:=Speck_tmp2[1].[10];
   		Speck_Rotate_Result[1].[12]:=Speck_tmp2[1].[9];
   		Speck_Rotate_Result[1].[11]:=Speck_tmp2[1].[8];
   		Speck_Rotate_Result[1].[10]:=Speck_tmp2[1].[7];
   		Speck_Rotate_Result[1].[9]:=Speck_tmp2[1].[6];
   		Speck_Rotate_Result[1].[8]:=Speck_tmp2[1].[5];
   		Speck_Rotate_Result[1].[7]:=Speck_tmp2[1].[4];
   		Speck_Rotate_Result[1].[6]:=Speck_tmp2[1].[3];
   		Speck_Rotate_Result[1].[5]:=Speck_tmp2[1].[2];
   		Speck_Rotate_Result[1].[4]:=Speck_tmp2[1].[1];
   		Speck_Rotate_Result[1].[3]:=Speck_tmp2[1].[0];
   		Speck_Rotate_Result[1].[2]:=Speck_tmp2[0].[31];
   		Speck_Rotate_Result[1].[1]:=Speck_tmp2[0].[30];
   		Speck_Rotate_Result[1].[0]:=Speck_tmp2[0].[29];
   		Speck_Rotate_Result[0].[31]:=Speck_tmp2[0].[28];
   		Speck_Rotate_Result[0].[30]:=Speck_tmp2[0].[27];
   		Speck_Rotate_Result[0].[29]:=Speck_tmp2[0].[26];
   		Speck_Rotate_Result[0].[28]:=Speck_tmp2[0].[25];
   		Speck_Rotate_Result[0].[27]:=Speck_tmp2[0].[24];
   		Speck_Rotate_Result[0].[26]:=Speck_tmp2[0].[23];
   		Speck_Rotate_Result[0].[25]:=Speck_tmp2[0].[22];
   		Speck_Rotate_Result[0].[24]:=Speck_tmp2[0].[21];
   		Speck_Rotate_Result[0].[23]:=Speck_tmp2[0].[20];
   		Speck_Rotate_Result[0].[22]:=Speck_tmp2[0].[19];
   		Speck_Rotate_Result[0].[21]:=Speck_tmp2[0].[18];
   		Speck_Rotate_Result[0].[20]:=Speck_tmp2[0].[17];
   		Speck_Rotate_Result[0].[19]:=Speck_tmp2[0].[16];
   		Speck_Rotate_Result[0].[18]:=Speck_tmp2[0].[15];
   		Speck_Rotate_Result[0].[17]:=Speck_tmp2[0].[14];
   		Speck_Rotate_Result[0].[16]:=Speck_tmp2[0].[13];
   		Speck_Rotate_Result[0].[15]:=Speck_tmp2[0].[12];
   		Speck_Rotate_Result[0].[14]:=Speck_tmp2[0].[11];
   		Speck_Rotate_Result[0].[13]:=Speck_tmp2[0].[10];
   		Speck_Rotate_Result[0].[12]:=Speck_tmp2[0].[9];
   		Speck_Rotate_Result[0].[11]:=Speck_tmp2[0].[8];
   		Speck_Rotate_Result[0].[10]:=Speck_tmp2[0].[7];
   		Speck_Rotate_Result[0].[9]:=Speck_tmp2[0].[6];
   		Speck_Rotate_Result[0].[8]:=Speck_tmp2[0].[5];
   		Speck_Rotate_Result[0].[7]:=Speck_tmp2[0].[4];
   		Speck_Rotate_Result[0].[6]:=Speck_tmp2[0].[3];
   		Speck_Rotate_Result[0].[5]:=Speck_tmp2[0].[2];
   		Speck_Rotate_Result[0].[4]:=Speck_tmp2[0].[1];
   		Speck_Rotate_Result[0].[3]:=Speck_tmp2[0].[0];
   End_CASE;
   
END_ROUTINE

ROUTINE SPECK_Rotate_Right_Dec   (* structured text *)
   Speck_Rotate_Result[0]:=0;
   Speck_Rotate_Result[1]:=0;
   
   CASE Speck_Ver Of
   	0:
   		Speck_Rotate_Result[0].[13]:=Speck_tmp2[0].[15];
   		Speck_Rotate_Result[0].[12]:=Speck_tmp2[0].[14];
   		Speck_Rotate_Result[0].[11]:=Speck_tmp2[0].[13];
   		Speck_Rotate_Result[0].[10]:=Speck_tmp2[0].[12];
   		Speck_Rotate_Result[0].[9]:=Speck_tmp2[0].[11];
   		Speck_Rotate_Result[0].[8]:=Speck_tmp2[0].[10];
   		Speck_Rotate_Result[0].[7]:=Speck_tmp2[0].[9];
   		Speck_Rotate_Result[0].[6]:=Speck_tmp2[0].[8];
   		Speck_Rotate_Result[0].[5]:=Speck_tmp2[0].[7];
   		Speck_Rotate_Result[0].[4]:=Speck_tmp2[0].[6];
   		Speck_Rotate_Result[0].[3]:=Speck_tmp2[0].[5];
   		Speck_Rotate_Result[0].[2]:=Speck_tmp2[0].[4];
   		Speck_Rotate_Result[0].[1]:=Speck_tmp2[0].[3];
   		Speck_Rotate_Result[0].[0]:=Speck_tmp2[0].[2];
   		Speck_Rotate_Result[0].[15]:=Speck_tmp2[0].[1];
   		Speck_Rotate_Result[0].[14]:=Speck_tmp2[0].[0];
   	1,2:
   		Speck_Rotate_Result[0].[28]:=Speck_tmp2[0].[31];
   		Speck_Rotate_Result[0].[27]:=Speck_tmp2[0].[30];
   		Speck_Rotate_Result[0].[26]:=Speck_tmp2[0].[29];
   		Speck_Rotate_Result[0].[25]:=Speck_tmp2[0].[28];
   		Speck_Rotate_Result[0].[24]:=Speck_tmp2[0].[27];
   		Speck_Rotate_Result[0].[23]:=Speck_tmp2[0].[26];
   		Speck_Rotate_Result[0].[22]:=Speck_tmp2[0].[25];
   		Speck_Rotate_Result[0].[21]:=Speck_tmp2[0].[24];
   		Speck_Rotate_Result[0].[20]:=Speck_tmp2[0].[23];
   		Speck_Rotate_Result[0].[19]:=Speck_tmp2[0].[22];
   		Speck_Rotate_Result[0].[18]:=Speck_tmp2[0].[21];
   		Speck_Rotate_Result[0].[17]:=Speck_tmp2[0].[20];
   		Speck_Rotate_Result[0].[16]:=Speck_tmp2[0].[19];
   		Speck_Rotate_Result[0].[15]:=Speck_tmp2[0].[18];
   		Speck_Rotate_Result[0].[14]:=Speck_tmp2[0].[17];
   		Speck_Rotate_Result[0].[13]:=Speck_tmp2[0].[16];
   		Speck_Rotate_Result[0].[12]:=Speck_tmp2[0].[15];
   		Speck_Rotate_Result[0].[11]:=Speck_tmp2[0].[14];
   		Speck_Rotate_Result[0].[10]:=Speck_tmp2[0].[13];
   		Speck_Rotate_Result[0].[9]:=Speck_tmp2[0].[12];
   		Speck_Rotate_Result[0].[8]:=Speck_tmp2[0].[11];
   		Speck_Rotate_Result[0].[7]:=Speck_tmp2[0].[10];
   		Speck_Rotate_Result[0].[6]:=Speck_tmp2[0].[9];
   		Speck_Rotate_Result[0].[5]:=Speck_tmp2[0].[8];
   		Speck_Rotate_Result[0].[4]:=Speck_tmp2[0].[7];
   		Speck_Rotate_Result[0].[3]:=Speck_tmp2[0].[6];
   		Speck_Rotate_Result[0].[2]:=Speck_tmp2[0].[5];
   		Speck_Rotate_Result[0].[1]:=Speck_tmp2[0].[4];
   		Speck_Rotate_Result[0].[0]:=Speck_tmp2[0].[3];
   		Speck_Rotate_Result[0].[31]:=Speck_tmp2[0].[2];
   		Speck_Rotate_Result[0].[30]:=Speck_tmp2[0].[1];
   		Speck_Rotate_Result[0].[29]:=Speck_tmp2[0].[0];
   	3,4,5:
   		Speck_Rotate_Result[1].[28]:=Speck_tmp2[1].[31];
   		Speck_Rotate_Result[1].[27]:=Speck_tmp2[1].[30];
   		Speck_Rotate_Result[1].[26]:=Speck_tmp2[1].[29];
   		Speck_Rotate_Result[1].[25]:=Speck_tmp2[1].[28];
   		Speck_Rotate_Result[1].[24]:=Speck_tmp2[1].[27];
   		Speck_Rotate_Result[1].[23]:=Speck_tmp2[1].[26];
   		Speck_Rotate_Result[1].[22]:=Speck_tmp2[1].[25];
   		Speck_Rotate_Result[1].[21]:=Speck_tmp2[1].[24];
   		Speck_Rotate_Result[1].[20]:=Speck_tmp2[1].[23];
   		Speck_Rotate_Result[1].[19]:=Speck_tmp2[1].[22];
   		Speck_Rotate_Result[1].[18]:=Speck_tmp2[1].[21];
   		Speck_Rotate_Result[1].[17]:=Speck_tmp2[1].[20];
   		Speck_Rotate_Result[1].[16]:=Speck_tmp2[1].[19];
   		Speck_Rotate_Result[1].[15]:=Speck_tmp2[1].[18];
   		Speck_Rotate_Result[1].[14]:=Speck_tmp2[1].[17];
   		Speck_Rotate_Result[1].[13]:=Speck_tmp2[1].[16];
   		Speck_Rotate_Result[1].[12]:=Speck_tmp2[1].[15];
   		Speck_Rotate_Result[1].[11]:=Speck_tmp2[1].[14];
   		Speck_Rotate_Result[1].[10]:=Speck_tmp2[1].[13];
   		Speck_Rotate_Result[1].[9]:=Speck_tmp2[1].[12];
   		Speck_Rotate_Result[1].[8]:=Speck_tmp2[1].[11];
   		Speck_Rotate_Result[1].[7]:=Speck_tmp2[1].[10];
   		Speck_Rotate_Result[1].[6]:=Speck_tmp2[1].[9];
   		Speck_Rotate_Result[1].[5]:=Speck_tmp2[1].[8];
   		Speck_Rotate_Result[1].[4]:=Speck_tmp2[1].[7];
   		Speck_Rotate_Result[1].[3]:=Speck_tmp2[1].[6];
   		Speck_Rotate_Result[1].[2]:=Speck_tmp2[1].[5];
   		Speck_Rotate_Result[1].[1]:=Speck_tmp2[1].[4];
   		Speck_Rotate_Result[1].[0]:=Speck_tmp2[1].[3];
   		Speck_Rotate_Result[0].[31]:=Speck_tmp2[1].[2];
   		Speck_Rotate_Result[0].[30]:=Speck_tmp2[1].[1];
   		Speck_Rotate_Result[0].[29]:=Speck_tmp2[1].[0];
   		Speck_Rotate_Result[0].[28]:=Speck_tmp2[0].[31];
   		Speck_Rotate_Result[0].[27]:=Speck_tmp2[0].[30];
   		Speck_Rotate_Result[0].[26]:=Speck_tmp2[0].[29];
   		Speck_Rotate_Result[0].[25]:=Speck_tmp2[0].[28];
   		Speck_Rotate_Result[0].[24]:=Speck_tmp2[0].[27];
   		Speck_Rotate_Result[0].[23]:=Speck_tmp2[0].[26];
   		Speck_Rotate_Result[0].[22]:=Speck_tmp2[0].[25];
   		Speck_Rotate_Result[0].[21]:=Speck_tmp2[0].[24];
   		Speck_Rotate_Result[0].[20]:=Speck_tmp2[0].[23];
   		Speck_Rotate_Result[0].[19]:=Speck_tmp2[0].[22];
   		Speck_Rotate_Result[0].[18]:=Speck_tmp2[0].[21];
   		Speck_Rotate_Result[0].[17]:=Speck_tmp2[0].[20];
   		Speck_Rotate_Result[0].[16]:=Speck_tmp2[0].[19];
   		Speck_Rotate_Result[0].[15]:=Speck_tmp2[0].[18];
   		Speck_Rotate_Result[0].[14]:=Speck_tmp2[0].[17];
   		Speck_Rotate_Result[0].[13]:=Speck_tmp2[0].[16];
   		Speck_Rotate_Result[0].[12]:=Speck_tmp2[0].[15];
   		Speck_Rotate_Result[0].[11]:=Speck_tmp2[0].[14];
   		Speck_Rotate_Result[0].[10]:=Speck_tmp2[0].[13];
   		Speck_Rotate_Result[0].[9]:=Speck_tmp2[0].[12];
   		Speck_Rotate_Result[0].[8]:=Speck_tmp2[0].[11];
   		Speck_Rotate_Result[0].[7]:=Speck_tmp2[0].[10];
   		Speck_Rotate_Result[0].[6]:=Speck_tmp2[0].[9];
   		Speck_Rotate_Result[0].[5]:=Speck_tmp2[0].[8];
   		Speck_Rotate_Result[0].[4]:=Speck_tmp2[0].[7];
   		Speck_Rotate_Result[0].[3]:=Speck_tmp2[0].[6];
   		Speck_Rotate_Result[0].[2]:=Speck_tmp2[0].[5];
   		Speck_Rotate_Result[0].[1]:=Speck_tmp2[0].[4];
   		Speck_Rotate_Result[0].[0]:=Speck_tmp2[0].[3];
   		Speck_Rotate_Result[1].[31]:=Speck_tmp2[0].[2];
   		Speck_Rotate_Result[1].[30]:=Speck_tmp2[0].[1];
   		Speck_Rotate_Result[1].[29]:=Speck_tmp2[0].[0];
   End_CASE;
   
END_ROUTINE

ROUTINE SPECK_Rotate_Right_Enc   (* structured text *)
   Speck_Rotate_Result[0]:=0;
   Speck_Rotate_Result[1]:=0;
   
   CASE Speck_Ver Of
   	0:
   		Speck_Rotate_Result[0].[8]:=Speck_tmp2[0].[15];
   		Speck_Rotate_Result[0].[7]:=Speck_tmp2[0].[14];
   		Speck_Rotate_Result[0].[6]:=Speck_tmp2[0].[13];
   		Speck_Rotate_Result[0].[5]:=Speck_tmp2[0].[12];
   		Speck_Rotate_Result[0].[4]:=Speck_tmp2[0].[11];
   		Speck_Rotate_Result[0].[3]:=Speck_tmp2[0].[10];
   		Speck_Rotate_Result[0].[2]:=Speck_tmp2[0].[9];
   		Speck_Rotate_Result[0].[1]:=Speck_tmp2[0].[8];
   		Speck_Rotate_Result[0].[0]:=Speck_tmp2[0].[7];
   		Speck_Rotate_Result[0].[15]:=Speck_tmp2[0].[6];
   		Speck_Rotate_Result[0].[14]:=Speck_tmp2[0].[5];
   		Speck_Rotate_Result[0].[13]:=Speck_tmp2[0].[4];
   		Speck_Rotate_Result[0].[12]:=Speck_tmp2[0].[3];
   		Speck_Rotate_Result[0].[11]:=Speck_tmp2[0].[2];
   		Speck_Rotate_Result[0].[10]:=Speck_tmp2[0].[1];
   		Speck_Rotate_Result[0].[9]:=Speck_tmp2[0].[0];
   	1,2:
   		Speck_Rotate_Result[0].[23]:=Speck_tmp2[0].[31];
   		Speck_Rotate_Result[0].[22]:=Speck_tmp2[0].[30];
   		Speck_Rotate_Result[0].[21]:=Speck_tmp2[0].[29];
   		Speck_Rotate_Result[0].[20]:=Speck_tmp2[0].[28];
   		Speck_Rotate_Result[0].[19]:=Speck_tmp2[0].[27];
   		Speck_Rotate_Result[0].[18]:=Speck_tmp2[0].[26];
   		Speck_Rotate_Result[0].[17]:=Speck_tmp2[0].[25];
   		Speck_Rotate_Result[0].[16]:=Speck_tmp2[0].[24];
   		Speck_Rotate_Result[0].[15]:=Speck_tmp2[0].[23];
   		Speck_Rotate_Result[0].[14]:=Speck_tmp2[0].[22];
   		Speck_Rotate_Result[0].[13]:=Speck_tmp2[0].[21];
   		Speck_Rotate_Result[0].[12]:=Speck_tmp2[0].[20];
   		Speck_Rotate_Result[0].[11]:=Speck_tmp2[0].[19];
   		Speck_Rotate_Result[0].[10]:=Speck_tmp2[0].[18];
   		Speck_Rotate_Result[0].[9]:=Speck_tmp2[0].[17];
   		Speck_Rotate_Result[0].[8]:=Speck_tmp2[0].[16];
   		Speck_Rotate_Result[0].[7]:=Speck_tmp2[0].[15];
   		Speck_Rotate_Result[0].[6]:=Speck_tmp2[0].[14];
   		Speck_Rotate_Result[0].[5]:=Speck_tmp2[0].[13];
   		Speck_Rotate_Result[0].[4]:=Speck_tmp2[0].[12];
   		Speck_Rotate_Result[0].[3]:=Speck_tmp2[0].[11];
   		Speck_Rotate_Result[0].[2]:=Speck_tmp2[0].[10];
   		Speck_Rotate_Result[0].[1]:=Speck_tmp2[0].[9];
   		Speck_Rotate_Result[0].[0]:=Speck_tmp2[0].[8];
   		Speck_Rotate_Result[0].[31]:=Speck_tmp2[0].[7];
   		Speck_Rotate_Result[0].[30]:=Speck_tmp2[0].[6];
   		Speck_Rotate_Result[0].[29]:=Speck_tmp2[0].[5];
   		Speck_Rotate_Result[0].[28]:=Speck_tmp2[0].[4];
   		Speck_Rotate_Result[0].[27]:=Speck_tmp2[0].[3];
   		Speck_Rotate_Result[0].[26]:=Speck_tmp2[0].[2];
   		Speck_Rotate_Result[0].[25]:=Speck_tmp2[0].[1];
   		Speck_Rotate_Result[0].[24]:=Speck_tmp2[0].[0];
   	3,4,5:
   		Speck_Rotate_Result[1].[23]:=Speck_tmp2[1].[31];
   		Speck_Rotate_Result[1].[22]:=Speck_tmp2[1].[30];
   		Speck_Rotate_Result[1].[21]:=Speck_tmp2[1].[29];
   		Speck_Rotate_Result[1].[20]:=Speck_tmp2[1].[28];
   		Speck_Rotate_Result[1].[19]:=Speck_tmp2[1].[27];
   		Speck_Rotate_Result[1].[18]:=Speck_tmp2[1].[26];
   		Speck_Rotate_Result[1].[17]:=Speck_tmp2[1].[25];
   		Speck_Rotate_Result[1].[16]:=Speck_tmp2[1].[24];
   		Speck_Rotate_Result[1].[15]:=Speck_tmp2[1].[23];
   		Speck_Rotate_Result[1].[14]:=Speck_tmp2[1].[22];
   		Speck_Rotate_Result[1].[13]:=Speck_tmp2[1].[21];
   		Speck_Rotate_Result[1].[12]:=Speck_tmp2[1].[20];
   		Speck_Rotate_Result[1].[11]:=Speck_tmp2[1].[19];
   		Speck_Rotate_Result[1].[10]:=Speck_tmp2[1].[18];
   		Speck_Rotate_Result[1].[9]:=Speck_tmp2[1].[17];
   		Speck_Rotate_Result[1].[8]:=Speck_tmp2[1].[16];
   		Speck_Rotate_Result[1].[7]:=Speck_tmp2[1].[15];
   		Speck_Rotate_Result[1].[6]:=Speck_tmp2[1].[14];
   		Speck_Rotate_Result[1].[5]:=Speck_tmp2[1].[13];
   		Speck_Rotate_Result[1].[4]:=Speck_tmp2[1].[12];
   		Speck_Rotate_Result[1].[3]:=Speck_tmp2[1].[11];
   		Speck_Rotate_Result[1].[2]:=Speck_tmp2[1].[10];
   		Speck_Rotate_Result[1].[1]:=Speck_tmp2[1].[9];
   		Speck_Rotate_Result[1].[0]:=Speck_tmp2[1].[8];
   		Speck_Rotate_Result[0].[31]:=Speck_tmp2[1].[7];
   		Speck_Rotate_Result[0].[30]:=Speck_tmp2[1].[6];
   		Speck_Rotate_Result[0].[29]:=Speck_tmp2[1].[5];
   		Speck_Rotate_Result[0].[28]:=Speck_tmp2[1].[4];
   		Speck_Rotate_Result[0].[27]:=Speck_tmp2[1].[3];
   		Speck_Rotate_Result[0].[26]:=Speck_tmp2[1].[2];
   		Speck_Rotate_Result[0].[25]:=Speck_tmp2[1].[1];
   		Speck_Rotate_Result[0].[24]:=Speck_tmp2[1].[0];
   		Speck_Rotate_Result[0].[23]:=Speck_tmp2[0].[31];
   		Speck_Rotate_Result[0].[22]:=Speck_tmp2[0].[30];
   		Speck_Rotate_Result[0].[21]:=Speck_tmp2[0].[29];
   		Speck_Rotate_Result[0].[20]:=Speck_tmp2[0].[28];
   		Speck_Rotate_Result[0].[19]:=Speck_tmp2[0].[27];
   		Speck_Rotate_Result[0].[18]:=Speck_tmp2[0].[26];
   		Speck_Rotate_Result[0].[17]:=Speck_tmp2[0].[25];
   		Speck_Rotate_Result[0].[16]:=Speck_tmp2[0].[24];
   		Speck_Rotate_Result[0].[15]:=Speck_tmp2[0].[23];
   		Speck_Rotate_Result[0].[14]:=Speck_tmp2[0].[22];
   		Speck_Rotate_Result[0].[13]:=Speck_tmp2[0].[21];
   		Speck_Rotate_Result[0].[12]:=Speck_tmp2[0].[20];
   		Speck_Rotate_Result[0].[11]:=Speck_tmp2[0].[19];
   		Speck_Rotate_Result[0].[10]:=Speck_tmp2[0].[18];
   		Speck_Rotate_Result[0].[9]:=Speck_tmp2[0].[17];
   		Speck_Rotate_Result[0].[8]:=Speck_tmp2[0].[16];
   		Speck_Rotate_Result[0].[7]:=Speck_tmp2[0].[15];
   		Speck_Rotate_Result[0].[6]:=Speck_tmp2[0].[14];
   		Speck_Rotate_Result[0].[5]:=Speck_tmp2[0].[13];
   		Speck_Rotate_Result[0].[4]:=Speck_tmp2[0].[12];
   		Speck_Rotate_Result[0].[3]:=Speck_tmp2[0].[11];
   		Speck_Rotate_Result[0].[2]:=Speck_tmp2[0].[10];
   		Speck_Rotate_Result[0].[1]:=Speck_tmp2[0].[9];
   		Speck_Rotate_Result[0].[0]:=Speck_tmp2[0].[8];
   		Speck_Rotate_Result[1].[31]:=Speck_tmp2[0].[7];
   		Speck_Rotate_Result[1].[30]:=Speck_tmp2[0].[6];
   		Speck_Rotate_Result[1].[29]:=Speck_tmp2[0].[5];
   		Speck_Rotate_Result[1].[28]:=Speck_tmp2[0].[4];
   		Speck_Rotate_Result[1].[27]:=Speck_tmp2[0].[3];
   		Speck_Rotate_Result[1].[26]:=Speck_tmp2[0].[2];
   		Speck_Rotate_Result[1].[25]:=Speck_tmp2[0].[1];
   		Speck_Rotate_Result[1].[24]:=Speck_tmp2[0].[0];
   End_CASE;
   
END_ROUTINE

ROUTINE SPECK_Sub   (* structured text *)
   Speck_AS_res[0]:=0;
   Speck_AS_res[1]:=0;
   
   	//big substraction low-32-bit
   		Speck_Sign_Bits[0].[0]:= Speck_AS_X[0].29; //keep the sign bit for big addition
   		Speck_Sign_Bits[0].[1]:= Speck_AS_X[0].30; //keep the sign bit for big addition
   		Speck_Sign_Bits[0].[2]:= Speck_AS_X[0].31; //keep the sign bit for big addition
   
   		Speck_AS_X[0].29:=0;
   		Speck_AS_X[0].30 :=1;   //give x  a 'virtual' borrow bit
   		Speck_AS_X[0].31:=0;
   
   
   
   		Speck_Sign_Bits[1].[0]:= Speck_AS_Y[0].29;
   		Speck_Sign_Bits[1].[1]:= Speck_AS_Y[0].30; //keep the sign bit for big addition
   		Speck_Sign_Bits[1].[2]:= Speck_AS_Y[0].31;
   		Speck_AS_Y[0].31:=0;
   		Speck_AS_Y[0].30:=0;
   		Speck_AS_Y[0].29:=0;
   
   		Speck_AS_res[0] := Speck_AS_X[0]-Speck_AS_Y[0];
   
   		Speck_Carry_Bit.[0]:= NOT Speck_AS_res[0].30;
   
   		Speck_Sign_Bits[0].[4]:=1;  //to ensure that Sign_Bits[0]> Sign_Bits[1]
   		Speck_AS_tmp:=Speck_Sign_Bits[0]-Speck_Sign_Bits[1]-Speck_Carry_Bit;
   
   
   
   		Speck_Carry_Bit.[0] := Speck_AS_tmp.[3];
   		Speck_AS_res[0].29:= Speck_AS_tmp.[0];
   		Speck_AS_res[0].30:= Speck_AS_tmp.[1];
   		Speck_AS_res[0].31:= Speck_AS_tmp.[2];
   
   
   		Speck_AS_tmp:=0;
   	 	Speck_Sign_Bits[0]:=0;
   	 	Speck_Sign_Bits[1]:=0;
   
   If Speck_Ver>2 Then
   
   		//sub high 32-bit
   
   		Speck_Sign_Bits[0].[0]:= Speck_AS_X[1].29; //keep the sign bit for big addition
   		Speck_Sign_Bits[0].[1]:= Speck_AS_X[1].30; //keep the sign bit for big addition
   		Speck_Sign_Bits[0].[2]:= Speck_AS_X[1].31; //keep the sign bit for big addition
   
   		Speck_AS_X[1].29:=0;
   		Speck_AS_X[1].30 :=1;   //give x  a 'virtual' borrow bit
   		Speck_AS_X[1].31:=0;
   
   
   
   		Speck_Sign_Bits[1].[0]:= Speck_AS_Y[1].29;
   		Speck_Sign_Bits[1].[1]:= Speck_AS_Y[1].30; //keep the sign bit for big addition
   		Speck_Sign_Bits[1].[2]:= Speck_AS_Y[1].31;
   		Speck_AS_Y[1].31:=0;
   		Speck_AS_Y[1].30:=0;
   		Speck_AS_Y[1].29:=0;
   
   		Speck_AS_res[1] := Speck_AS_X[1]-Speck_AS_Y[1] -Speck_Carry_Bit;
   
   		Speck_Carry_Bit.[0]:= NOT Speck_AS_res[1].30;
   
   		Speck_Sign_Bits[0].[4]:=1;
   		Speck_AS_tmp:=Speck_Sign_Bits[0]-Speck_Sign_Bits[1]-Speck_Carry_Bit;
   
   
   
   		Speck_AS_res[1].29:= Speck_AS_tmp.[0];
   		Speck_AS_res[1].30:= Speck_AS_tmp.[1];
   		Speck_AS_res[1].31:= Speck_AS_tmp.[2];
   
   End_If;
   
   
   		//clear
   		Speck_Carry_Bit:=0;
   		Speck_AS_tmp:=0;
   		Speck_Sign_Bits[0]:=0;
   		Speck_Sign_Bits[1]:=0;
   		Speck_AS_X[0]:=0;
   		Speck_AS_X[1]:=0;
   		Speck_AS_Y[0]:=0;
   		Speck_AS_Y[1]:=0;
   
END_ROUTINE
END_PROGRAM
